FUNCTION_BLOCK CylinderHCore (* Ground-truth reference: continuous-time cylinder position model (E_CYCLE tick + integEC integrator + ChangeDetect filter) *)
  (* Standard: 61499-2; Description: Educational reference, ported for the Meisterschulen am Ostbahnhof IEC 61499 training repository. Original design (c) nxtControl GmbH, from the UniversalAutomation.org 'IEC 61499: primer course' curriculum exercise Final.sln (also present in the LiftingLuggage_*.sln/Starter.sln exercises), IEC61499/CylinderH/CylinderH.fbt - included here under the same educational-use terms as the rest of that curriculum. This port: Copyright (c) 2026 Meisterschulen am Ostbahnhof, EPL-2.0, https://www.eclipse.org/legal/epl-2.0/ *)
  (* Version 0.0, 2016-05-25, Andrei, nxtControl GmbH, Original EAE/nxtControl design (Template), source: Final.sln (identical copies in LiftingLuggage_*.sln, Starter.sln), original name CylinderH *)
  (* Version 1.0, 2026-09-03, Franz Höpfinger, Meisterschulen am Ostbahnhof, Core-only port: renamed CylinderH -> CylinderHCore. Dropped LABEL (display-only) and the CylinderH_HMI instance (a native Service Interface FB with no portable ECC/algorithm - just a QI/QO init passthrough plus an HMI display, not part of the physical model) and replaced its structural role (relaying INITO onward to start the E_CYCLE ticker and to this block's own INTO) with a direct connection. Uses the standard iec61499::events::E_CYCLE instead of porting a duplicate - see the check-standard-lib-before-creating lesson. integEC/ChangeDetect otherwise unchanged, see ContinuousCylinderSimulation.md *)
  (* Version 1.1, 2026-09-03, Franz Höpfinger, Meisterschulen am Ostbahnhof, PR #160 review feedback: INIT/INITO must be Type=EInit (were Type=Event) - fixed; renamed the init-confirm event from INTO to INITO to match this repo's convention (Copilot review comment). Also restored the E_CYCLE Import declaration, which had gone empty. *)
  (* Version 1.2, 2026-09-03, Franz Höpfinger, Meisterschulen am Ostbahnhof, PR #160 review feedback (coderabbitai): a repeated INIT, sent after the cylinder had already moved, forwarded Model.INITO to Tick.START/INITO without first updating Filter, so POSITION still showed the stale pre-reset value instead of the freshly-reset 0.0. Fixed by also wiring Model.INITO -> Filter.REQ, declared before the other two INITO fan-out connections so Filter.OUT/POSITION update first *)
  PACKAGE Meins::DesingPatterns::ContinuousCylinderSimulation;
  (* Documentation:
  Ground-truth reference, not a Vyatkin Module 6 slide pattern. Core-only port of the UniversalAutomation.org "IEC 61499: primer course" curriculum's CylinderH (Final.sln, IEC61499/CylinderH/CylinderH.fbt - identical copies exist in the LiftingLuggage_*.sln/Starter.sln exercises, and it is itself the innermost layer of the CylinderHSens/CylinderHSensValve composites seen there). A genuinely different modelling technique from this repo's EventDrivenCylinder.fbt/CylinderService.fbt (Purely-Event-Driven pattern / slide-47 message-exchange example): those are discrete event-driven state machines with zero continuous data; this is a continuous-time physics simulation - an E_CYCLE ticks every 20 ms, driving integEC (a generic time-based integrator) to ramp a REAL POSITION value between 0.0 (retracted) and 130.0 (extended) based on the PV1/PV2 drive signals, filtered through ChangeDetect so IND only fires when the position actually moved. INIT/INITO use Type="EInit" (fixed from the original port's Type="Event" and the original event name INTO, renamed to INITO to match this repo's convention - PR #160 review feedback). Matches the "Modelling Event-driven PLCs system" / "Modelling a Scan-based PLCs System" slides (Module 6, slides 50-52) more closely than any pattern actually implemented in this repo so far - found while searching the curriculum for material relevant to already-implemented patterns, kept here as its own standalone reference rather than folded into an existing pattern folder.
   Reduced vs. the original (by explicit choice, not full fidelity): dropped the LABEL display string and the CylinderH_HMI instance - a native EAE Service Interface FB (Interface1 in the original) with no portable ECC/algorithm of its own, just a QI/QO init passthrough plus an HMI panel. Its one structural role - relaying Model.INITO onward to start the E_CYCLE ticker and to this block's own INITO - is preserved here as a direct connection instead. See CylinderH_HMI.fbt/CylinderHSens.fbt/ CylinderHSensValve.fbt in the original curriculum export for the full chain (sensor wrapping, valve control, HMI) if a more complete port is ever needed.
  *)
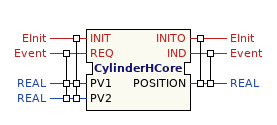
  EVENT_INPUT
    INIT : EInit WITH PV1, PV2; (* Initialization Request *)
    REQ WITH PV1, PV2; (* Normal Execution Request: apply new PV1/PV2 drive signals *)
  END_EVENT
  EVENT_OUTPUT
    INITO : EInit WITH POSITION; (* Initialization Confirm *)
    IND WITH POSITION; (* Position changed *)
  END_EVENT
  VAR_INPUT
    PV1 : REAL; (* Extend drive signal, fed to integEC.pv1 *)
    PV2 : REAL; (* Retract drive signal (inverted), fed to integEC.pv2 *)
  END_VAR
  VAR_OUTPUT
    POSITION : REAL; (* Current cylinder position, 0.0 (retracted) to 130.0 (extended) *)
  END_VAR
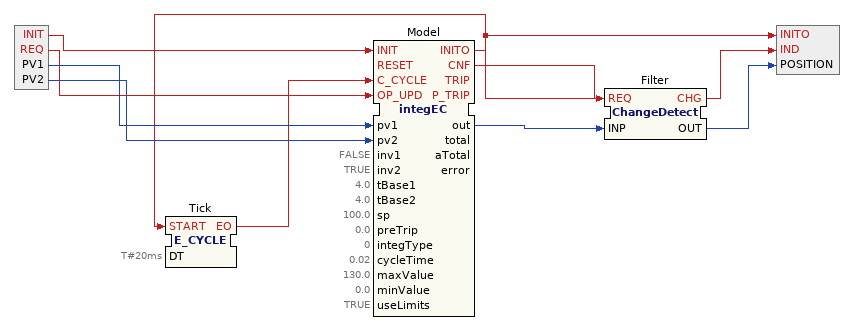
  FBS
    Tick : iec61499::events::E_CYCLE(DT := T#20ms);
    Model : Meins::DesingPatterns::ContinuousCylinderSimulation::integEC(inv1 := FALSE, inv2 := TRUE, tBase1 := 4.0, tBase2 := 4.0, sp := 100.0, preTrip := 0.0, integType := 0, cycleTime := 0.02, maxValue := 130.0, minValue := 0.0, useLimits := TRUE);
    Filter : Meins::DesingPatterns::ContinuousCylinderSimulation::ChangeDetect;
  END_FBS
  EVENT_CONNECTIONS
    INIT TO Model.INIT;
    Model.INITO TO Filter.REQ;
    Model.INITO TO Tick.START;
    Model.INITO TO INITO;
    Tick.EO TO Model.C_CYCLE;
    REQ TO Model.OP_UPD;
    Model.CNF TO Filter.REQ;
    Filter.CHG TO IND;
  END_CONNECTIONS
  DATA_CONNECTIONS
    PV1 TO Model.pv1;
    PV2 TO Model.pv2;
    Model.out TO Filter.INP;
    Filter.OUT TO POSITION;
  END_CONNECTIONS
END_FUNCTION_BLOCK
